// TIA Portal V20 export
// export: Created 2026-10-03T18:54:34.2836607Z, ExportSetting WithDefaults, DisplayName Totally Integrated Automation Portal, DisplayVersion V20 Update 4, DisplayName TIA Portal Openness, DisplayVersion V20 Update 4, DisplayName TIA Portal Version Control Interface, DisplayVersion V20 Update 4, DisplayName SINAMICS Startdrive Advanced, DisplayVersion V20 SP1 Update 1, DisplayName SINAMICS Startdrive G110M, G120, G120C, G120D, G120P, G115D, DisplayVersion V20 SP1 Update 1, DisplayName SINAMICS Startdrive G130, G150, S120, S150, SINAMICS MV, G220, S200, S210, DisplayVersion V20 SP1 Update 1, DisplayName STEP 7 Professional, DisplayVersion V20 Update 4, DisplayName STEP 7 Safety, DisplayVersion V20 Update 2, DisplayName WinCC Basic/Comfort/Advanced, DisplayVersion V20 Update 4, DisplayName WinCC Unified, DisplayVersion V20 Update 4
FUNCTION "SLC_FLL_FLOAT" : Void   // FC13, SCL
TITLE = SLC FLL (fill file) for F files
{ S7_Optimized_Access := 'TRUE' }
VERSION : 0.1
// Replaces FLL Value #DstFile:DstElement Length for floating point files.
// stored: AutoNumber true, IsIECCheckEnabled false, SetENOAutomatically false, UDAEnableTagReadback false
   VAR_INPUT
      Value : Real;   // Value to fill with
      DstFile : DInt;   // Destination data file number
      DstElement : DInt;   // First element to fill
      Length : DInt;   // Number of elements to fill
   END_VAR
   VAR_TEMP
      i : DInt;
   END_VAR
BEGIN
   FOR #i := 0 TO #Length - 1 DO
       // 16#84 is the DB memory area; each element is 4 bytes.
       POKE(area := 16#84, dbNumber := #DstFile, byteOffset := (#DstElement + #i) * 4, value := #Value);
   END_FOR;
END_FUNCTION
